{attribute 'qualified_only'}
{attribute 'strict'}
{attribute 'to_string'}
TYPE E_RobotCommandState :
(
    Idle := 0,
    Requested := 1,
    Sending := 2,
    Accepted := 3,
    Executing := 4,
    Done := 5,
    Aborted := 6,
    Error := 7
);
END_TYPE

(* stored: Version 1.1.0.1, ProductVersion 3.1.4026.18
   DUT E_RobotCommandState: Id {b8b8fd7b-9879-4c58-95b4-ced43300d1fb} *)
